PROGRAM MAIN
VAR
END_VAR

EmgFunctions();

END_PROGRAM

(* stored: Version 1.1.0.1, ProductVersion 3.1.4024.9
   POU MAIN: Id {6be4bdac-14e8-49dd-bc56-eb748116da27}, SpecialFunc None *)
